{attribute 'GeneratedUsingTerminal: EK1122-0000-0018'}
{attribute addProperty BoxType "EK1122-0000-0018"}
{attribute addProperty Id "Beckhoff_APS1xxxsub_EK1100EK1100_1FC0878B2A_0001_APS1003_7000_0016APS1003_4F8F3E0B256"}
{attribute addProperty CRC "3439946889"}
{attribute addProperty Size "258"}
TYPE Beckhoff_APS1xxxEK1122_CD096C89 EXTENDS EK1122_1FC0878B :
STRUCT
	{attribute addProperty Name "Beckhoff_APS1xxxsub_EK1100"}
	{attribute addProperty PreviousPort "Beckhoff APS1xxxEK1122 : D"}
	Beckhoff_APS1xxxsub_EK1100 : EK1100_1FC0878B;
	{attribute addProperty Name "A_0001_APS1003_7000_0016"}
	{attribute addProperty PreviousPort "Beckhoff APS1xxxsub EK1100 : C"}
	A_0001_APS1003_7000_0016 : APS1003_4F8F3E0B;
END_STRUCT
END_TYPE

(* stored: Version 1.2.0.0, ProductVersion 3.1.4024.9
   DUT Beckhoff_APS1xxxEK1122_CD096C89: Id {ac4e3622-ffdb-43d5-baa7-6e6fce83c13e} *)
